FUNCTION_BLOCK PAProcessModule EXTENDS PAClassPhysicalBase IMPLEMENTS IPAProcessModule 
VAR_INPUT
END_VAR
VAR_OUTPUT
END_VAR
VAR
	_Allocated : BOOL;
END_VAR

{attribute 'monitoring' := 'call'}
{attribute 'TcRpcEnable'}
PROPERTY PUBLIC Allocated : BOOL
GET
Allocated := _Allocated;
END_GET
SET
_Allocated := Allocated;
Root.OnPropertyChangedBool(THIS^, 16, _Allocated);
END_SET
END_PROPERTY

METHOD PUBLIC FB_postinit
VAR_INPUT
		root : IACVariobatch;
END_VAR
SUPER^.FB_postinit(root);
Root.OnPropertyChangedBool(THIS^, 16, _Allocated);
END_METHOD

METHOD PROTECTED GetRoutingStateOfDependents  : PARoutingState
VAR_INPUT
	controlModule	: IPAControlModule;
	rStateAll : PARoutingState;
	direction : PARoutingDirection;
END_VAR
VAR
	activePF : IPAProcessFunction;
	currentPF : IPAProcessFunction;
	i: INT;
END_VAR
activePF := controlModule.AllocatedByFunction;

// Suche nach aktiver Prozessfunktion, die in diesem Prozessmodul vorliegt
// Es müssen keine Points durchsucht werden, da normalerweise ein Ein-/Ausgangspunkt eine Prozessmodules immer mit einem Punkt einer Prozessfunktion verbunden sein sollte
// (eine Edge vom Typ LogicalBrige)
IF activePF = 0 THEN
	GetRoutingStateOfDependents := PARoutingState.Idle;
	RETURN;
END_IF

GetRoutingStateOfDependents := PARoutingState.Idle;
FOR i:=1 TO GCL.cChildsMAX BY 1
  DO
    IF (_Childs[i] <> 0) THEN
		IF __QUERYINTERFACE(_Childs[i], currentPF) THEN
			IF activePF = currentPF THEN
				// Falls gefunden gebe einfach den aktuellen Routingstatus, des Vorgänger-ControlModuls zurück.
				GetRoutingStateOfDependents := rStateAll;
				RETURN;
			END_IF
		END_IF
	ELSE
		EXIT;
	END_IF
END_FOR;
END_METHOD

METHOD OnInitMemory
VAR_INPUT
	root : IACVariobatch;
END_VAR
RegisterProperty(root, 16, GCL.cSizeBYTE); //Allocated
SUPER^.OnInitMemory(root);
END_METHOD

METHOD RoutingStateFromSource : PARoutingState
VAR_INPUT
	controlModule: IPAControlModule;
	rStateAll : PARoutingState;
END_VAR
RoutingStateFromSource := GetRoutingStateOfDependents(controlModule, rStateAll, PARoutingDirection.ToPredecessors);
END_METHOD

METHOD RoutingStateToTarget : PARoutingState
VAR_INPUT
	controlModule: IPAControlModule;
	rStateAll : PARoutingState;
END_VAR
RoutingStateToTarget := GetRoutingStateOfDependents(controlModule, rStateAll, PARoutingDirection.ToSuccessors);
END_METHOD

END_FUNCTION_BLOCK

(* stored: Version 1.1.0.1, ProductVersion 3.1.4024.6
   POU PAProcessModule: Id {6c01c64c-a15e-4232-b69d-0c8e44fa854b}, SpecialFunc None
   Property Allocated: Id {bea17035-c899-4924-a5d9-29cbf433a68f}
   Get Get: Id {32a211e0-f30e-4643-8fa4-a6fa241b0818}
   Set Set: Id {2b52d50c-fe0e-4248-9f68-4132a6409b52}
   Method FB_postinit: Id {fc896cbe-d39a-468b-b7d9-ab016e66809d}
   Method GetRoutingStateOfDependents: Id {ec89391f-b555-43fb-b295-065ef60c0e38}
   Method OnInitMemory: Id {3ea7b46c-1da6-41d8-9160-5bebd163629e}
   Method RoutingStateFromSource: Id {675129f3-a06f-4e98-9837-0aabe2afa9c1}
   Method RoutingStateToTarget: Id {6747f9a9-f260-4cf1-9945-bc34f6727062} *)
